# EPICS substitutions: db/Beckhoff_1XXX/ecmcEL1859.substitutions
# binary inputs
file "ecmc_binaryInput-chX.template"{
  pattern {CH_ID}
          {01   }
          {02   }
          {03   }
          {04   }
          {05   }
          {06   }
          {07   }
          {08   }
}

file "ecmc_binaryOutput-chX.template"
{
  pattern {CH_ID}
          {01   }
          {02   }
          {03   }
          {04   }
          {05   }
          {06   }
          {07   }
          {08   }
}
